(* CoDeSys 2.3.9.35 project: Exercicio1 - 1 - mais certo.pro *)
(* Author: d *)
(* Libraries: DU35x.lib 26.11.09 14:36:14, Navigation.lib 2.6.09 12:09:20, SysLibTargetVisu.lib 26.11.08 09:53:28, Standard.lib 26.11.08 09:46:20, Iecsfc.lib 26.11.08 09:46:14, SYSLIBCALLBACK.LIB 26.11.08 09:53:30 *)

(* PLC configuration (modules and I/O channels)
Comunicação [Comunica] node 0, in %IB0 out %QB0
  COM1 [COM1] node 0, in %IB0 out %QB0 {BaudRate = 115200; Paridade = Sem Paridade; StopBits = 1 Stop Bit; Modem = Sem RTS/CTS; Delay = 5}
    MToolIEC [Codesys] node 0, in %IB0 out %QB0
  COM2 [COM2] node 1, in %IB0 out %QB0 {BaudRate = 115200; Paridade = Sem Paridade; StopBits = 1 Stop Bit; Modem = Sem RTS/CTS; Delay = 5}
    Desabilitada [Desabilitado485] node 0, in %IB0 out %QB0
Entradas Digitais 0 [Entradas0] node 0, in %IW0 out %QB0
  I00 AT %IX0.0 [BitInput] I0.0
  I01 AT %IX0.1 [BitInput] I0.1
  I02 AT %IX0.2 [BitInput] I0.2
  I03 AT %IX0.3 [BitInput] I0.3
  I04 AT %IX0.4 [BitInput] I0.4
  I05 AT %IX0.5 [BitInput] I0.5
  I06 AT %IX0.6 [BitInput] I0.6
  I07 AT %IX0.7 [BitInput] I0.7
  I08 AT %IX0.8 [BitInput] I0.8
Entradas Digitais 1 [Entradas1] node 0, in %IW1 out %QB0
  I10 AT %IX1.0 [BitInput] I1.0
  I11 AT %IX1.1 [BitInput] I1.1
  I12 AT %IX1.2 [BitInput] I1.2
  I13 AT %IX1.3 [BitInput] I1.3
  I14 AT %IX1.4 [BitInput] I1.4
  I15 AT %IX1.5 [BitInput] I1.5
  I16 AT %IX1.6 [BitInput] I1.6
  I17 AT %IX1.7 [BitInput] I1.7
  I18 AT %IX1.8 [BitInput] I1.8
Entradas Digitais 2 [Entradas2] node 0, in %IW2 out %QB0
  I20 AT %IX2.0 [BitInput] I2.0
  I21 AT %IX2.1 [BitInput] I2.1
AI0 AT %IW4 [WordInput] AI0 {TipoAnalogica = Tensão 0-10V; FiltroAnalogica = Filtro 0 - AI=2ms  / AV=90ms; FundoEscala = 1000}
AI1 AT %IW5 [WordInput] AI1 {TipoAnalogica = Canal Desabilitado; FiltroAnalogica = Filtro 0 - AI=2ms  / AV=90ms; FundoEscala = 0}
AI2 AT %IW6 [WordInput] AI2 {TipoAnalogica = Canal Desabilitado; FiltroAnalogica = Filtro 0 - AI=2ms  / AV=90ms; FundoEscala = 0}
AI3 AT %IW7 [WordInput] AI3 {TipoAnalogica = Canal Desabilitado; FiltroAnalogica = Filtro 0 - AI=2ms  / AV=90ms; FundoEscala = 0}
Entradas Rápidas [EntradasRapidas] node 1, in %IB16 out %QB0
  Bloco 0 [Bloco0] node 0, in %IB16 out %QB0
    Desabilitado [DesabilitadoBloco0] node 0, in %IB16 out %QB0
  Bloco 1 [Bloco1] node 1, in %IB16 out %QB0
    Desabilitado [DesabilitadoBloco1] node 0, in %IB16 out %QB0
  Entrada Configuravél Bloco 0 [EntradaConfiBloco0] node 2, in %IB16 out %QB0
    Contador 0 [EntradaConfContador0] node 0, in %IB16 out %QB0 {EntradaConfiguravelContador = Desabilitada}
  Entrada Configuravél Bloco 1 [EntradaConfiBloco1] node 3, in %IB16 out %QB0
    Contador 2 [EntradaConfContador2] node 0, in %IB16 out %QB0 {EntradaConfiguravelContador = Desabilitada}
Saídas [Saidas] node 1, in %IB13 out %QB0
  Saídas Digitais 0 [Saidas0] node 0, in %IW0 out %QW0
    Q00 AT %QX0.0 [BitOutput] Q0.0
    Q01 AT %QX0.1 [BitOutput] Q0.1
    Q02 AT %QX0.2 [BitOutput] Q0.2
    Q03 AT %QX0.3 [BitOutput] Q0.3
    Q04 AT %QX0.4 [BitOutput] Q0.4
    Q05 AT %QX0.5 [BitOutput] Q0.5
    Q06 AT %QX0.6 [BitOutput] Q0.6
    Q07 AT %QX0.7 [BitOutput] Q0.7
  Saídas Digitais 1 [Saidas1] node 0, in %IW0 out %QW1
    Q10 AT %QX1.0 [BitOutput] Q1.0
    Q11 AT %QX1.1 [BitOutput] Q1.1
    Q12 AT %QX1.2 [BitOutput] Q1.2
    Q13 AT %QX1.3 [BitOutput] Q1.3
    Q14 AT %QX1.4 [BitOutput] Q1.4
    Q15 AT %QX1.5 [BitOutput] Q1.5
    Q16 AT %QX1.6 [BitOutput] Q1.6
    Q17 AT %QX1.7 [BitOutput] Q1.7
  Saídas Analógicas [SaidaAnalogica] node 0, in %IW0 out %QW3
    AO0 AT %QW3 [WordOutput] AO0 {TipoAnalogica = Canal Desabilitado; FundoEscala = 0}
    AO1 AT %QW4 [WordOutput] AO1 {TipoAnalogica = Canal Desabilitado; FundoEscala = 0}
  Saídas Rápidas [SaidasRapidas] node 1, in %IB0 out %QB10
    Saída Rápida 0 Desabilitada [DesabilitadoF0] node 0, in %IB0 out %QB10
    Saída Rápida 1 Desabilitada [DesabilitadoF1] node 1, in %IB0 out %QB10
  Saídas Comum de Contador [SaidasContador] node 2, in %IB0 out %QB10
    Saída do Bloco 0 Desabilitada [DesabilitadoSaidaBloco0] node 0, in %IB0 out %QB10
    Saída do Bloco 1 Desabilitada [DesabilitadoSaidaBloco1] node 1, in %IB0 out %QB10
Eventos Externos [Eventos] node 2, in %IB13 out %QB6
  Evento Temporizado [TimerEvent] node 0, in %IB13 out %QB6 {Intervalo = 10}
*)

(* Task configuration *)
TASK PRINCIPAL (PRIORITY := 1, INTERVAL := T#1ms);
	PLC_PRG();
END_TASK
TASK NAVIGATION (PRIORITY := 1, INTERVAL := T#20ms);
	NAVEGA();
END_TASK
TASK VISUALIZATION (PRIORITY := 1, INTERVAL := T#500ms);
	MAINTARGETVISU_PAINT_CODE
END_TASK
TASK KEYBOARD_USAGE (PRIORITY := 1, INTERVAL := T#20ms);
	MAINTARGETVISU_INPUT_CODE
END_TASK

(* POU PLC_PRG, LD *)
(*Elabore um comando liga-desliga utilizando como comando a entrada analógica. Acione a carga quando a tensão de entrada for
inferior um limite MIN (valor inicial de 4,00 V) e desligue a carga quando a tensão de entrada for superior a um limite MAX 
(valor inicial de 6,00 V). Os valores MAX e MIN devem poder ser editados pela IHM. Caso um botão de EMERGENCIA seja acionado 
a qualquer instante, a carga deve ser imediatamente desligada, e um novo acionamento só poderá ser realizado após o sinal de 
entrada permanecer por, no mínimo, 10s em 0V. Exiba o valor de tensão lido na IHM, em 3 telas diferentes, utilizando elementos
gráficos diferentes. Usar a escala apropriada (duas casa decimais) e com indicação de unidade.*)

PROGRAM PLC_PRG
VAR
	DL AT %IX0.0: BOOL;
	S1 AT %QX1.0: BOOL;
	T1: TON;
    M1: BOOL;
    BS1: F_TRIG;
    AN AT %IW4: WORD;
	AN_REAL: REAL;
	M2: BOOL;
	VMIN: REAL:=4.0;
    VMAX: REAL:=6.0;
	M3: BOOL;
	M4: BOOL;
	M5: BOOL;
	M6: BOOL;
	M7: BOOL;
	M8: BOOL;
END_VAR
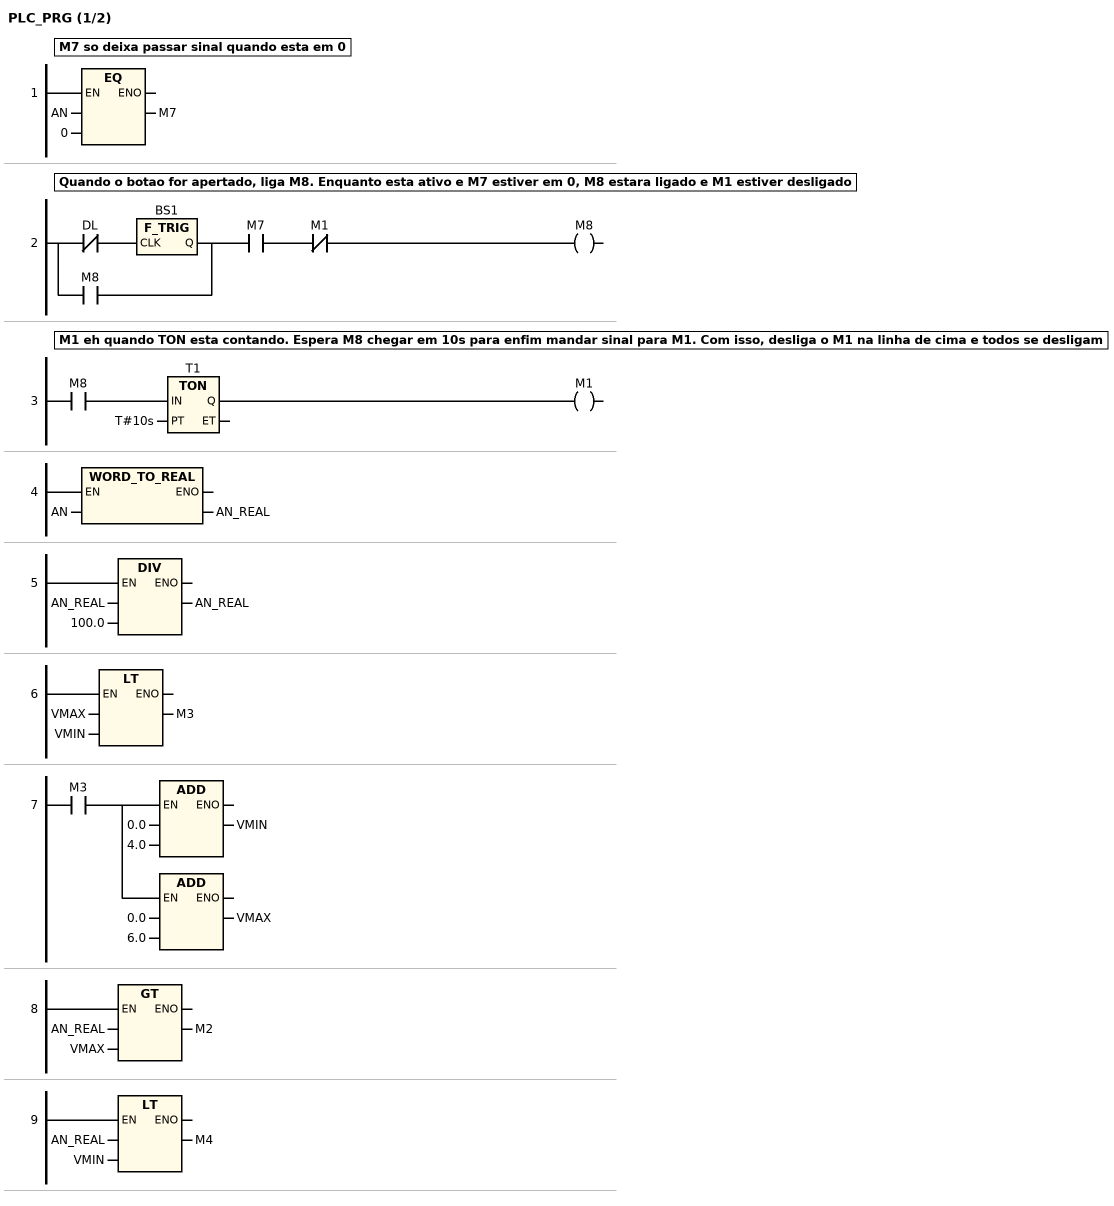
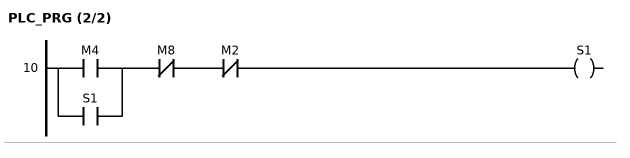
_LD_ (* Ladder Diagram *)
NETWORK 1 M7 so deixa passar sinal quando esta em 0:
	*
		EN --- EQ(AN, 0) => M7
NETWORK 2 Quando o botao for apertado, liga M8. Enquanto esta ativo e M7 estiver em 0, M8 estara ligado e M1 estiver desligado:
	{ [/DL] - BS1:F_TRIG(CLK: *) | [M8] } - [M7] - [/M1] --- (M8)
NETWORK 3 M1 eh quando TON esta contando. Espera M8 chegar em 10s para enfim mandar sinal para M1. Com isso, desliga o M1 na linha de cima e todos se desligam:
	[M8] - T1:TON(IN: *, PT: T#10s) --- (M1)
NETWORK 4
	*
		EN --- WORD_TO_REAL(AN) => AN_REAL
NETWORK 5
	*
		EN --- DIV(AN_REAL, 100.0) => AN_REAL
NETWORK 6
	*
		EN --- LT(VMAX, VMIN) => M3
NETWORK 7
	[M3]
		EN --- ADD(0.0, 4.0) => VMIN
		EN --- ADD(0.0, 6.0) => VMAX
NETWORK 8
	*
		EN --- GT(AN_REAL, VMAX) => M2
NETWORK 9
	*
		EN --- LT(AN_REAL, VMIN) => M4
NETWORK 10
	{ [M4] | [S1] } - [/M8] - [/M2] --- (S1)
_END_LD_
(* the same logic as Structured Text *)
(* Network 1 *)
(* label: M7 so deixa passar sinal quando esta em 0 *)
M7 := AN = 0;
(* Network 2 *)
(* label: Quando o botao for apertado, liga M8. Enquanto esta ativo e M7 estiver em 0, M8 estara ligado e M1 estiver desligado *)
BS1(CLK := NOT DL);
M8 := (BS1.Q OR M8) AND M7 AND NOT M1;
(* Network 3 *)
(* label: M1 eh quando TON esta contando. Espera M8 chegar em 10s para enfim mandar sinal para M1. Com isso, desliga o M1 na linha de cima e todos se desligam *)
T1(IN := M8, PT := T#10s);
M1 := T1.Q;
(* Network 4 *)
AN_REAL := WORD_TO_REAL(AN);
(* Network 5 *)
AN_REAL := AN_REAL / 100.0;
(* Network 6 *)
M3 := VMAX < VMIN;
(* Network 7 *)
IF M3 THEN
	VMIN := 0.0 + 4.0;
	VMAX := 0.0 + 6.0;
END_IF;
(* Network 8 *)
M2 := AN_REAL > VMAX;
(* Network 9 *)
M4 := AN_REAL < VMIN;
(* Network 10 *)
S1 := (M4 OR S1) AND NOT M8 AND NOT M2;
END_PROGRAM

(* POU NAVEGA, ST *)
PROGRAM NAVEGA
VAR
	ControleTelas : NAVIGATION;
	ListaTelas 	: ARRAY [0..30] OF STRING(10);
	CONTRASTE AT %MB6468 : BYTE; (* Percentagem do contraste *)
	BACKLIGHT AT %MB6469 : BYTE; (* Configuração do backlight *)
END_VAR
(* Contraste do display em 40% *)
CONTRASTE := 40;
(* Desliga o backlight quando ficar 30 segundos oscioso *)
BACKLIGHT := 30;

(* Adiciona a tela MAIN como tela principal *)
ListaTelas[0] := 'MAIN';

(* Ativa o controle automático de navegação somente pelo teclado *)
ControleTelas(ENABLE_UPDW := FALSE, VISU_LIST := ListaTelas, UP := FALSE , DOWN := FALSE);
END_PROGRAM

(* Visualisation MAIN
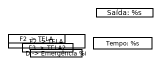
rectangle at (68,4)-(125,13): text "Saída: %s"; shows PLC_PRG.S1
rectangle at (-20,30)-(37,39): text "F2 -> TELA"
rectangle at (65,33)-(124,45): text "Tempo: %s"; shows PLC_PRG.T1.ET
rectangle at (-20,30)-(57,44): text "F2 -> TELA"
rectangle at (-6,39)-(45,48): text "F3 -> TELA2"
rectangle at (2,45)-(54,53): text "D -> Emergência %i"; shows PLC_PRG.DL
4 elements of other kinds (tables, trends, ...) not read
*)

(* Visualisation TELA
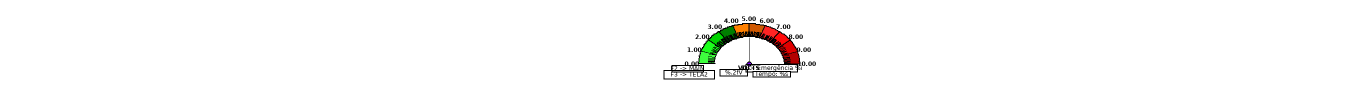
group at (15,-2)-(143,55)
  rectangle at (0,0)-(1,1): text "{ExtendedElement},Visu\ElementDLL.ete,0,@Zeigerinstrument,144,180,0,3,128,0,255,0,PLC_PRG.AN_REAL,VOLTS,%.2f,0,1,1,0.1,1,0,10,0,0,0,0,0,0,0,-5,40,700,Arial,1,10,0,1,62,255,62,1,2,28,255,28,2,3,0,210,0,3,4,0,127,0,4,5,255,128,0,5,6,208,89,2,6,7,255,36,36,7,8,255,9,9,8,9,223,0,0,9,10,179,0,0,"
  rectangle at (3,69)-(13,75): text "0.00"
  rectangle at (6,49)-(16,55): text "1.00"
  rectangle at (15,31)-(25,37): text "2.00"
  rectangle at (29,17)-(39,23): text "3.00"
  rectangle at (47,8)-(57,14): text "4.00"
  rectangle at (67,5)-(77,11): text "5.00"
  rectangle at (87,8)-(97,14): text "6.00"
  rectangle at (105,17)-(115,23): text "7.00"
  rectangle at (119,31)-(129,37): text "8.00"
  rectangle at (128,49)-(138,55): text "9.00"
  rectangle at (130,69)-(143,75): text "10.00"
  rectangle at (64,75)-(80,81): text "VOLTS"
  polygon at (72,35)-(72,72): angle ((PLC_PRG.AN_REAL * 1.0)-5) * 18
rectangle at (50,54)-(78,61): text "%.2fV"; shows PLC_PRG.AN_REAL
rectangle at (2,50)-(34,57): text "F2 -> MAIN"
rectangle at (-6,55)-(45,64): text "F3 -> TELA2"
rectangle at (76,49)-(128,57): text "D -> Emergência %i"; shows PLC_PRG.DL
rectangle at (83,56)-(121,62): text "Tempo: %s"; shows PLC_PRG.T1.ET
114 more shapes without text or variables
*)

(* Visualisation TELA2
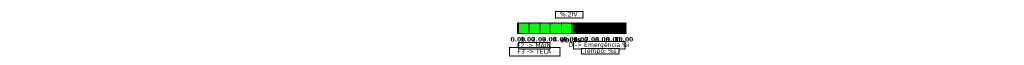
group at (6,14)-(125,60)
  rectangle at (0,0)-(1,1): text "{ExtendedElement},Visu\ElementDLL.ete,1,@Bargraph,119,46,1,0,0,PLC_PRG.AN_REAL,VOLTS,%.2f,1,1,0,10,0,0,0,0,0,0,0,-3,20,700,Arial,0,255,0,255,0,0,0,0,1,0,0,"
  rectangle at (7,8)-(60,16): alarm colour if (PLC_PRG.AN_REAL) < 0; right ((PLC_PRG.AN_REAL * 1.0) - 5)  * 10.4
  rectangle at (2,18)-(11,42): text "0.00"
  rectangle at (12,18)-(21,42): text "1.00"
  rectangle at (23,18)-(32,42): text "2.00"
  rectangle at (33,18)-(42,42): text "3.00"
  rectangle at (44,18)-(53,42): text "4.00"
  rectangle at (54,18)-(63,42): text "5.00"
  rectangle at (64,18)-(73,42): text "6.00"
  rectangle at (75,18)-(84,42): text "7.00"
  rectangle at (85,18)-(94,42): text "8.00"
  rectangle at (96,18)-(105,42): text "9.00"
  rectangle at (105,18)-(117,42): text "10.00"
  rectangle at (49,21)-(69,25): text "VOLTS"
rectangle at (13,41)-(45,48): text "F2 -> MAIN"
rectangle at (4,46)-(55,55): text "F3 -> TELA"
rectangle at (68,40)-(120,48): text "D -> Emergência %i"; shows PLC_PRG.DL
rectangle at (76,47)-(114,53): text "Tempo: %s"; shows PLC_PRG.T1.ET
rectangle at (50,10)-(78,17): text "%.2fV"; shows PLC_PRG.AN_REAL
12 more shapes without text or variables
*)
